// TIA Portal V21 export
DATA_BLOCK "Data_block_1"   // DB1
{ S7_Optimized_Access := 'TRUE' }
   VAR
      "zmienna 1" : Bool;
      "zmienna 2" : Bool;
   END_VAR
BEGIN
END_DATA_BLOCK
